{attribute 'qualified_only'}
VAR_GLOBAL
	nNumber1 : DINT;
END_VAR

(* stored: Version 1.1.0.1, ProductVersion 3.1.4024.16
   GVL GVL_Sum: Id {3e276d38-be3d-4dd2-974f-15a044cb1e36} *)
